SUBAPPLICATION PartPresenceSensor (* Subapplication Type *)
  (* Standard: 61499-2 *)
  (* Version 1.0, 2020-07-28, dummy *)
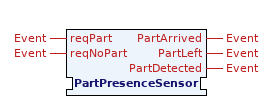
  EVENT_INPUT
    reqPart;
    reqNoPart;
  END_EVENT
  EVENT_OUTPUT
    PartArrived;
    PartLeft;
    PartDetected;
  END_EVENT
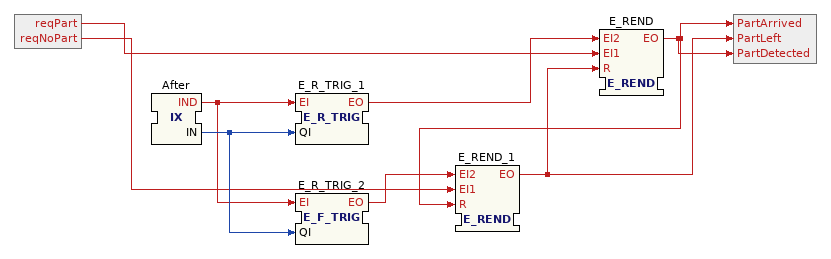
  FBS
    E_R_TRIG_1 : E_R_TRIG;
    After : IX;
    E_R_TRIG_2 : E_F_TRIG;
    E_REND : E_REND;
    E_REND_1 : E_REND;
  END_FBS
  EVENT_CONNECTIONS
    After.IND TO E_R_TRIG_1.EI;
    After.IND TO E_R_TRIG_2.EI;
    E_R_TRIG_1.EO TO E_REND.EI2;
    E_R_TRIG_2.EO TO E_REND_1.EI2;
    reqPart TO E_REND.EI1;
    reqNoPart TO E_REND_1.EI1;
    E_REND.EO TO E_REND_1.R;
    E_REND_1.EO TO E_REND.R;
    E_REND.EO TO PartArrived;
    E_REND_1.EO TO PartLeft;
    E_REND.EO TO PartDetected;
  END_CONNECTIONS
  DATA_CONNECTIONS
    After.IN TO E_R_TRIG_1.QI;
    After.IN TO E_R_TRIG_2.QI;
  END_CONNECTIONS
END_SUBAPPLICATION
